PROGRAM MAIN
VAR_OUTPUT
	localTime : TIMESTRUCT; //used by watchdogs, not set in module
END_VAR
VAR
	spacerRecollector : SpacerRecollectionUnit;
END_VAR
VAR
	robot7 : RobotA26;
	robotSliderA26 : ServoNC := (
		limitSensorDefaultState := TRUE,
		enableDualSideTraverse := TRUE);
		
END_VAR
VAR //sensors to detect spacers on receiver conveyors
	spacerPresent_A24_LRC_C02 AT %I* : BOOL;
	spacerPresent_A24_LRC_C04 AT %I* : BOOL;
	spacerPresent_A24_LRC_C06 AT %I* : BOOL;
	spacerPresent_A24_LRC_C08 AT %I* : BOOL;
	spacerPresent_A24_LRC_C10 AT %I* : BOOL;
	spacerPresent_A24_LRC_C12 AT %I* : BOOL;
END_VAR

CallHardware(); //start program with hardware call
SetupHardware(); //not applicable for this module

runModules();

CallHardware(); //end program with hardware call

METHOD PROTECTED callHardware : BOOL
VAR_INPUT
END_VAR
robot7(bEnable:= TRUE, abort:= , conveyorSafety:= TRUE);	
robotSliderA26(bEnable:= TRUE, ready=> , position=> , velocity=> );
END_METHOD

METHOD PROTECTED runModules : BOOL
VAR_INPUT
END_VAR
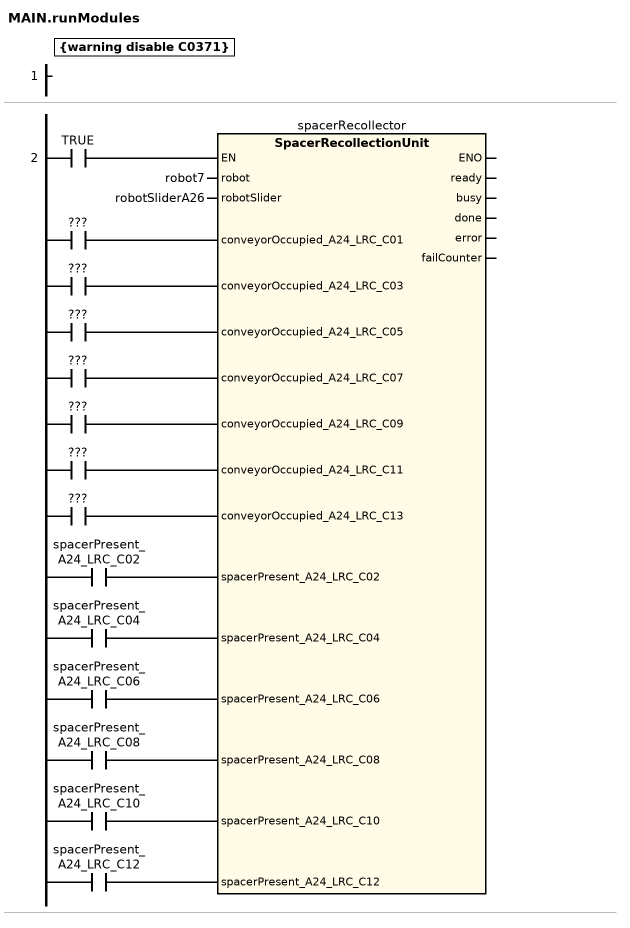
// NETWORK 1
// label: {warning disable C0371}

// NETWORK 2
spacerRecollector(
    robot := robot7,
    robotSlider := robotSliderA26,
    spacerPresent_A24_LRC_C02 := spacerPresent_A24_LRC_C02,
    spacerPresent_A24_LRC_C04 := spacerPresent_A24_LRC_C04,
    spacerPresent_A24_LRC_C06 := spacerPresent_A24_LRC_C06,
    spacerPresent_A24_LRC_C08 := spacerPresent_A24_LRC_C08,
    spacerPresent_A24_LRC_C10 := spacerPresent_A24_LRC_C10,
    spacerPresent_A24_LRC_C12 := spacerPresent_A24_LRC_C12); // SpacerRecollectionUnit
END_METHOD

METHOD PROTECTED setupHardware : BOOL
VAR
	
END_VAR
END_METHOD

END_PROGRAM

(* stored: Version 1.1.0.1, ProductVersion 3.1.4024.11
   POU MAIN: Id {67e6f294-cce3-4abb-aa77-8a640eacb7df}, SpecialFunc None
   Method callHardware: Id {28545458-26ff-4a6a-af8e-aff99ab2b072}
   Method runModules: Id {91fb3897-d479-41a4-ac07-1d36f5ff9718}
   Method setupHardware: Id {0b0eb0a5-de16-4ffc-920a-53d441a1c49c} *)
